FUNCTION_BLOCK AX_T_FF_SR_SEQ_GATE (* Wie AX_T_FF_SR_SEQ (echt bidirektional: 4 strikt getrennte Pfade Vorwaerts-Set/Vorwaerts-Reset/Rueckwaerts-Set/Rueckwaerts-Reset), zusaetzlich mit Freigabe-Socket GATE:AX und eigenem Zustand GATE_CLOSED - geht GATE auf FALSE, wird sofort zwangsweise RESET ausgefuehrt und in GATE_CLOSED gesperrt; einziger Ausweg aus GATE_CLOSED ist GATE.E1[GATE.D1] (Gate wieder offen) *)
  (* Standard: 61499-1 Annex A; Function: Wie AX_T_FF_SR_SEQ (lokales S/R/CLK, 4 strikt getrennte CHAIN-Pfade ueber ASR2: CHAIN_IN.EO_SET->CHAIN_OUT.EO_SET, CHAIN_IN.EO_RESET->CHAIN_OUT.EO_RESET, CHAIN_OUT.EI_SET->CHAIN_IN.EI_SET, CHAIN_OUT.EI_RESET->CHAIN_IN.EI_RESET - keine Verzweigung, jeder Zustand feuert genau eine Chain-Aktion), zusaetzlich: GATE (Socket, AX) muss TRUE sein, sonst wird der Baustein in einen eigenen Zustand GATE_CLOSED gezwungen (Q.E1 mit FALSE, wie RESET). In GATE_CLOSED ist S/R/CLK/CHAIN_IN/CHAIN_OUT komplett wirkungslos (keine Transition definiert - IEC 61499 verwirft das Event einfach) - der EINZIGE Ausweg ist GATE.E1[GATE.D1] zurueck nach RESET. Ein waehrend GATE_CLOSED ankommendes Chain-Event (vorwaerts oder rueckwaerts) wird NICHT weitergereicht - ein gesperrtes Kettenglied unterbricht die Kette fuer nachfolgende Glieder in beide Richtungen (bewusste, aber revisitierbare Designentscheidung). *)
  (* Version 1.4, 2026-09-17, Franz Höpfinger, HR Agrartechnik GmbH, Echte Bidirektionalitaet ergaenzt (Franz: 'Chain IN SET --> Chain Out Set, und Rueckwaerts auch so. keine Events verdoppeln... insgesamt 4 Pfade. keine Verzweigungen'), analog AX_T_FF_SR_SEQ v1.1: 2 neue Zustaende SET_CHAIN_BWD/RESET_CHAIN_BWD fuer die Rueckwaerts-Richtung (CHAIN_OUT.EI_SET/EI_RESET -> lokal + CHAIN_IN.EI_SET/EI_RESET), inkl. GATE-Pruefung [NOT GATE.D1] als erste Transition auch auf den beiden neuen Zustaenden - Rueckwaerts-Set wird durch GATE genauso gesperrt wie Vorwaerts-Set. *)
  (* Version 1.3, 2026-09-17, Franz Höpfinger, HR Agrartechnik GmbH, Bugfix (Reihenfolge-Luecke, analog AX_T_FF_SR_GATE): GATE.E1[NOT GATE.D1] durch ereignisloses [NOT GATE.D1] ersetzt UND in jedem Zustand an die ERSTE Stelle der Deklarationsreihenfolge gesetzt (vorher standen S/CLK/CHAIN_IN.EO_SET davor - da diese ohne Guard immer TRUE sind, hat IEC 61499-1 Table 1 Regel c) sie zuerst gekreuzt, die Gate-Sperre kam bei S/CLK/CHAIN_IN.EO_SET nie zum Zug). Doppelte START->GATE_CLOSED-Transition (Epsilon + event-getriggert) auf eine ereignislose Variante konsolidiert - deckt jetzt sowohl Boot-Fenster als auch laufendes Monitoring bei JEDEM Event ab (nicht nur GATE.E1), siehe DIN/EVS EN 61499-1 Table 1 Regel c4/c5. *)
  (* Version 1.1, 2026-09-17, Franz Höpfinger, HR Agrartechnik GmbH, Umgebaut (Franz: 'brauchen wir da nicht einen Zustand GATE_CLOSED? aus dem Zustand kommt man nur raus mit GATE.E1[GATE.D1 = TRUE]'): V1.0 hatte GATE.D1 als 12 verstreute [GATE.D1]-Guards auf jeder einzelnen EIN-Transition - funktional aequivalent, aber schwer auditierbar. Jetzt 1 dedizierter Zustand GATE_CLOSED: alle EIN-Transitionen wieder ungegatet (wie AX_T_FF_SR_SEQ), Sperre lebt ausschliesslich in GATE_CLOSEDs fehlenden Ausgangs-Transitionen fuer S/R/CLK/CHAIN_IN - deutlich einfacher zu verifizieren ('der einzige Weg raus ist die eine GATE.E1[GATE.D1]-Transition'). *)
  (* Version 1.0, 2026-09-17, Franz Höpfinger, HR Agrartechnik GmbH, Neu (Franz: 'mach gleich noch ein AX_T_FF_SR_SEQ_GATE was einen zusaetzlichen AX hat, der AN sein muss als Freigabe... wenn AX aus geht ist der Baustein gesperrt, es wird RESET ausgefuehrt. SET wird nur akzeptiert wenn das Gate wieder offen ist'). Kopiert von AX_T_FF_SR_SEQ. Loest das frueher zurueckgestellte FORCE_OFF-Problem ('haelt R durchgehend, aber Baustein geht dafuer nicht, sofortiges Wiedereinschalten moeglich') fuer den Zapfwellen-Ueberwachungs-Anwendungsfall: hier ist die Sperre echt pegelbasiert, kein reiner Flanken-Puls auf R. *)
  PACKAGE adapter::events::unidirectional;
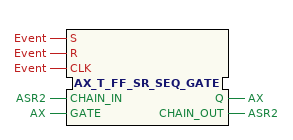
  EVENT_INPUT
    S; (* Set output Q (lokal, wirkt nie auf CHAIN_IN/CHAIN_OUT) - wirkungslos waehrend GATE_CLOSED *)
    R; (* Reset output Q (lokal, wirkt nie auf CHAIN_IN/CHAIN_OUT) - wirkungslos waehrend GATE_CLOSED (ist ohnehin schon aus) *)
    CLK; (* Clock for triggering a output toggle (lokal, wirkt nie auf CHAIN_IN/CHAIN_OUT) - wirkungslos waehrend GATE_CLOSED *)
  END_EVENT
  SOCKETS
    CHAIN_IN : adapter::types::bidirectional::ASR2; (* Vorwaerts: Set/Reset vom vorherigen Kettenglied empfangen (EO_SET/EO_RESET). Rueckwaerts: Set/Reset an vorheriges Kettenglied weiterreichen (EI_SET/EI_RESET). Nicht waehrend GATE_CLOSED. *)
    GATE : adapter::types::unidirectional::AX; (* Freigabe: muss TRUE sein. Faellt GATE auf FALSE: sofort GATE_CLOSED (Zwangs-RESET + Sperre), verlassen nur ueber GATE.E1[GATE.D1]. *)
  END_SOCKETS
  PLUGS
    Q : adapter::types::unidirectional::AX; (* value of flip flop *)
    CHAIN_OUT : adapter::types::bidirectional::ASR2; (* Vorwaerts: Set/Reset an naechstes Kettenglied (EO_SET/EO_RESET). Rueckwaerts: Set/Reset VOM naechsten Kettenglied empfangen (EI_SET/EI_RESET). Nicht waehrend GATE_CLOSED. *)
  END_PLUGS
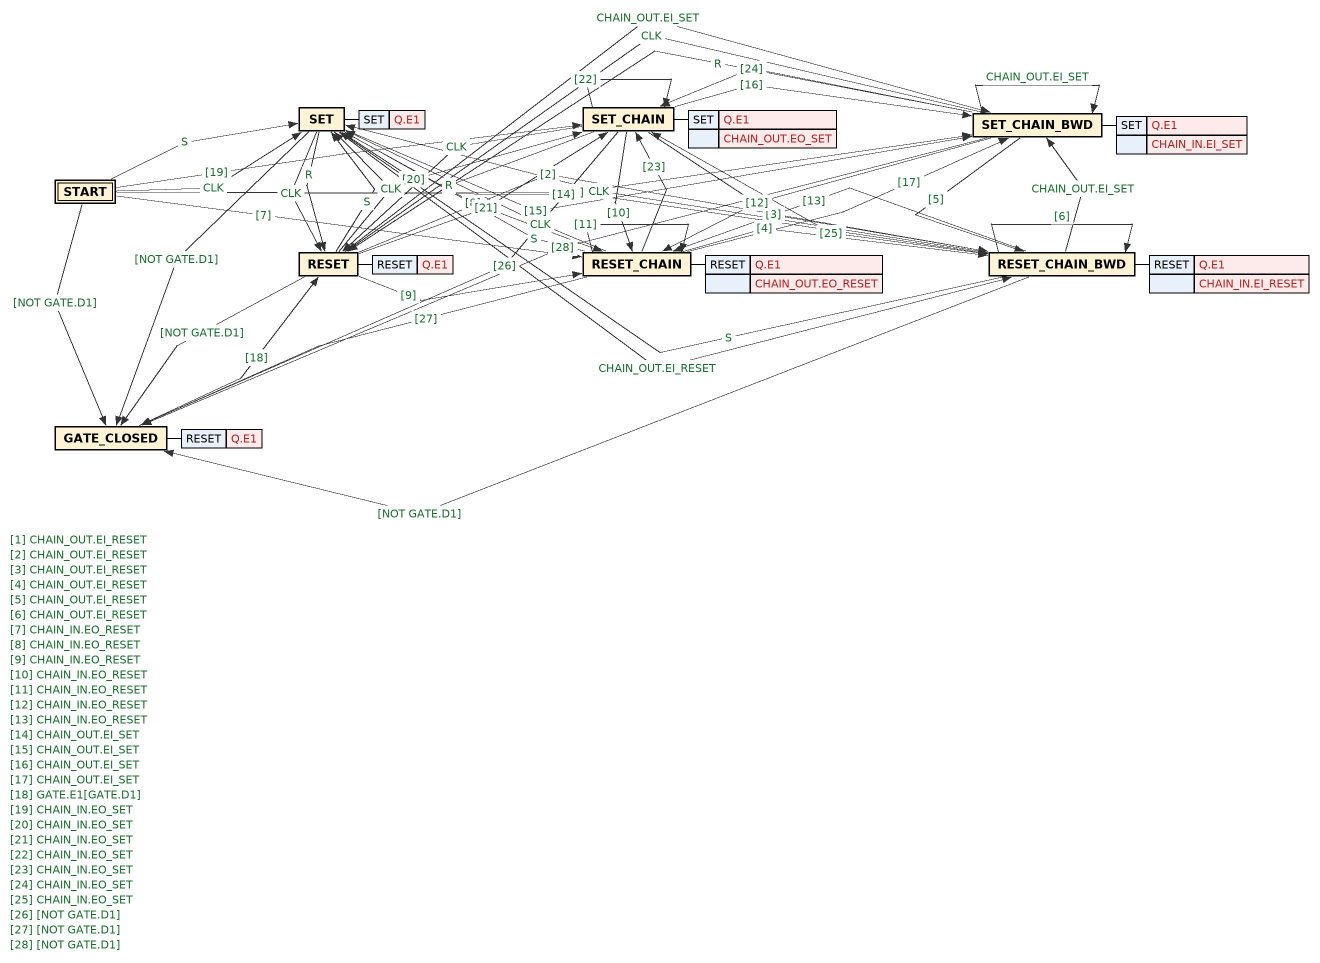
  EC_STATES
    START; (* Initial State *)
    SET : SET -> Q.E1;
    RESET : RESET -> Q.E1;
    SET_CHAIN : SET -> Q.E1, -> CHAIN_OUT.EO_SET; (* Set kam vorwaerts ueber CHAIN_IN.EO_SET - reicht NUR vorwaerts an CHAIN_OUT.EO_SET weiter *)
    RESET_CHAIN : RESET -> Q.E1, -> CHAIN_OUT.EO_RESET; (* Reset kam vorwaerts ueber CHAIN_IN.EO_RESET - reicht NUR vorwaerts an CHAIN_OUT.EO_RESET weiter *)
    SET_CHAIN_BWD : SET -> Q.E1, -> CHAIN_IN.EI_SET; (* Set kam rueckwaerts ueber CHAIN_OUT.EI_SET - reicht NUR rueckwaerts an CHAIN_IN.EI_SET weiter *)
    RESET_CHAIN_BWD : RESET -> Q.E1, -> CHAIN_IN.EI_RESET; (* Reset kam rueckwaerts ueber CHAIN_OUT.EI_RESET - reicht NUR rueckwaerts an CHAIN_IN.EI_RESET weiter *)
    GATE_CLOSED : RESET -> Q.E1; (* Gesperrt: GATE.D1=FALSE. Q zwangsweise FALSE. S/R/CLK/CHAIN_IN/CHAIN_OUT sind hier wirkungslos (keine Transition definiert). Einziger Ausweg: GATE.E1[GATE.D1] zurueck nach RESET. *)
  END_STATES
  EC_TRANSITIONS
    START TO GATE_CLOSED := [NOT GATE.D1];
    START TO SET := S;
    START TO SET := CLK;
    START TO SET_CHAIN := CHAIN_IN.EO_SET;
    START TO RESET_CHAIN := CHAIN_IN.EO_RESET;
    START TO SET_CHAIN_BWD := CHAIN_OUT.EI_SET;
    START TO RESET_CHAIN_BWD := CHAIN_OUT.EI_RESET;
    SET TO GATE_CLOSED := [NOT GATE.D1];
    SET TO RESET := R;
    SET TO RESET := CLK;
    SET TO SET_CHAIN := CHAIN_IN.EO_SET;
    SET TO RESET_CHAIN := CHAIN_IN.EO_RESET;
    SET TO SET_CHAIN_BWD := CHAIN_OUT.EI_SET;
    SET TO RESET_CHAIN_BWD := CHAIN_OUT.EI_RESET;
    RESET TO GATE_CLOSED := [NOT GATE.D1];
    RESET TO SET := S;
    RESET TO SET := CLK;
    RESET TO SET_CHAIN := CHAIN_IN.EO_SET;
    RESET TO RESET_CHAIN := CHAIN_IN.EO_RESET;
    RESET TO SET_CHAIN_BWD := CHAIN_OUT.EI_SET;
    RESET TO RESET_CHAIN_BWD := CHAIN_OUT.EI_RESET;
    SET_CHAIN TO GATE_CLOSED := [NOT GATE.D1];
    SET_CHAIN TO RESET := R;
    SET_CHAIN TO RESET := CLK;
    SET_CHAIN TO SET_CHAIN := CHAIN_IN.EO_SET;
    SET_CHAIN TO RESET_CHAIN := CHAIN_IN.EO_RESET;
    SET_CHAIN TO SET_CHAIN_BWD := CHAIN_OUT.EI_SET;
    SET_CHAIN TO RESET_CHAIN_BWD := CHAIN_OUT.EI_RESET;
    RESET_CHAIN TO GATE_CLOSED := [NOT GATE.D1];
    RESET_CHAIN TO SET := S;
    RESET_CHAIN TO SET := CLK;
    RESET_CHAIN TO SET_CHAIN := CHAIN_IN.EO_SET;
    RESET_CHAIN TO RESET_CHAIN := CHAIN_IN.EO_RESET;
    RESET_CHAIN TO SET_CHAIN_BWD := CHAIN_OUT.EI_SET;
    RESET_CHAIN TO RESET_CHAIN_BWD := CHAIN_OUT.EI_RESET;
    SET_CHAIN_BWD TO GATE_CLOSED := [NOT GATE.D1];
    SET_CHAIN_BWD TO RESET := R;
    SET_CHAIN_BWD TO RESET := CLK;
    SET_CHAIN_BWD TO SET_CHAIN := CHAIN_IN.EO_SET;
    SET_CHAIN_BWD TO RESET_CHAIN := CHAIN_IN.EO_RESET;
    SET_CHAIN_BWD TO SET_CHAIN_BWD := CHAIN_OUT.EI_SET;
    SET_CHAIN_BWD TO RESET_CHAIN_BWD := CHAIN_OUT.EI_RESET;
    RESET_CHAIN_BWD TO GATE_CLOSED := [NOT GATE.D1];
    RESET_CHAIN_BWD TO SET := S;
    RESET_CHAIN_BWD TO SET := CLK;
    RESET_CHAIN_BWD TO SET_CHAIN := CHAIN_IN.EO_SET;
    RESET_CHAIN_BWD TO RESET_CHAIN := CHAIN_IN.EO_RESET;
    RESET_CHAIN_BWD TO SET_CHAIN_BWD := CHAIN_OUT.EI_SET;
    RESET_CHAIN_BWD TO RESET_CHAIN_BWD := CHAIN_OUT.EI_RESET;
    GATE_CLOSED TO RESET := GATE.E1[GATE.D1];
  END_TRANSITIONS
  ALGORITHM SET IN ST:
Q.D1 := TRUE;
  END_ALGORITHM
  ALGORITHM RESET IN ST:
Q.D1 := FALSE;
  END_ALGORITHM
END_FUNCTION_BLOCK
